PROGRAM MAIN
VAR
	cleaningfb1: Cleaning;
END_VAR

IF gvl.CleanMachine = TRUE THEN 
	Cleaning(TypeCleaning := 1);
ELSIF gvl.Start = TRUE THEN 
	gvl.FillCup := TRUE;
END_IF

END_PROGRAM

(* stored: Version 1.1.0.1, ProductVersion 3.1.4024.12
   POU MAIN: Id {1d951c8b-fcff-4624-aa4d-0b666ca2df31}, SpecialFunc None *)
